{region "VFD"}
    //Status
    VTD_Control.Motor.Ready := (VTD_Control.Inputs.VFD_Status.%X0 OR VTD_Control.Inputs.VFD_Status.%X1) AND NOT VTD_Control.Motor.Error;
    VTD_Control.Motor.Error := VTD_Control.Inputs.VFD_Status.%X3 OR VTD_Control.Inputs.VFD_Status.%X7 OR NOT VTD_Control.Inputs.VFD_Status.%X13;
    VTD_Control.Motor.Enabled := VTD_Control.Inputs.VFD_Status.%X2;
    VTD_Control.Motor.Actual_Current := VTD_Control.Inputs.VFD_ActualCurrent;
    VTD_Control.Motor.Actual_Torque := SCALE_X(MIN := 0,
                                                VALUE := NORM_X(MIN := 0,
                                                                VALUE := VTD_Control.Inputs.VFD_ActualTorque,
                                                                MAX := 65536),
                                                MAX := 100);
    
    //Actual Speed
    IF MainSetpoint > 0 THEN
        VTD_Control.Motor.Speed_Actual := SCALE_X(MIN := 0,
                                                   VALUE := NORM_X(MIN := 0,
                                                                   VALUE := VTD_Control.Inputs.VFD_Speed_Actual,
                                                                   MAX := 16384),
                                                   MAX := 120);
        VTD_Control.Motor.Actual_Torque := SCALE_X(MIN := 0,
                                                    VALUE := NORM_X(MIN := 0,
                                                                    VALUE := VTD_Control.Inputs.VFD_ActualTorque * -1,
                                                                    MAX := 16384),
                                                    MAX := 100);
    ELSIF MainSetpoint < 0 THEN
        VTD_Control.Motor.Speed_Actual := SCALE_X(MIN := 0,
                                                   VALUE := NORM_X(MIN := 0,
                                                                   VALUE := VTD_Control.Inputs.VFD_Speed_Actual * -1,
                                                                   MAX := 16384),
                                                   MAX := 120);
        VTD_Control.Motor.Actual_Torque := SCALE_X(MIN := 0,
                                                    VALUE := NORM_X(MIN := 0,
                                                                    VALUE := VTD_Control.Inputs.VFD_ActualTorque * -1,
                                                                    MAX := 16384),
                                                    MAX := 100);
    ELSE
        VTD_Control.Motor.Speed_Actual := 0;
        VTD_Control.Motor.Actual_Torque := 0;
    END_IF;
    
    //SETPOINT
    IF VTD_Control.Motor_UP THEN
        MainSetpoint := SCALE_X(MIN := 0,
                                 VALUE := NORM_X(MIN := 0,
                                                 VALUE := VTD_Control.Motor_Speed,
                                                 MAX := 120),
                                 MAX := 1762);
    ELSIF VTD_Control.Motor_Down THEN
        MainSetpoint := (SCALE_X(MIN := 0,
                                  VALUE := NORM_X(MIN := 0,
                                                  VALUE := VTD_Control.Motor_Speed,
                                                  MAX := 120),
                                  MAX := 1762)) * -1;
    ELSE
        MainSetpoint := 0;
    END_IF;
    
    T_Setpoint_Delay(IN := MainSetpoint <> 0,
                          PT := T#0MS);
    
    IF T_Setpoint_Delay.Q THEN
        MainSetpoint1 := MainSetpoint;
    ELSE
        MainSetpoint1 := 0;
    END_IF;
    
    //Acceleration
    IF VTD_Control.Pallet_Loaded = 0 AND VTD_Control.Shuttle_Loaded = 0 THEN
        VTD_Control.Motor.Acc_Factor := SCALE_X(MIN := 0,
                                                 VALUE := NORM_X(MIN := 0,
                                                                 VALUE := 60.0,
                                                                 MAX := 100),
                                                 MAX := 16384);
    ELSIF Control.VTD_Order_Table[System_no].Pallet_Weight > 0 AND
        Control.VTD_Order_Table[System_no].Pallet_Weight <= "Settings_DB".VTD_Sys[System_no].Weight_Range_1 THEN
        VTD_Control.Motor.Acc_Factor := SCALE_X(MIN := 0,
                                                 VALUE := NORM_X(MIN := 0,
                                                                 VALUE := "Settings_DB".VTD_Sys[System_no].Acc_Range_1,
                                                                 MAX := 100),
                                                 MAX := 16384);
    ELSIF Control.VTD_Order_Table[System_no].Pallet_Weight > "Settings_DB".VTD_Sys[System_no].Weight_Range_1 AND
        Control_GVL.VTD_Order_Table[System_no].Pallet_Weight <= "Settings_DB".VTD_Sys[System_no].Weight_Range_2 THEN
        VTD_Control.Motor.Acc_Factor := SCALE_X(MIN := 0,
                                                 VALUE := NORM_X(MIN := 0,
                                                                 VALUE := "Settings_DB".VTD_Sys[System_no].Acc_Range_2,
                                                                 MAX := 100),
                                                 MAX := 16384);
    ELSIF Control.VTD_Order_Table[System_no].Pallet_Weight > "Settings_DB".VTD_Sys[System_no].Weight_Range_2 AND
        Control_GVL.VTD_Order_Table[System_no].Pallet_Weight <= "Settings_DB".VTD_Sys[System_no].Weight_Range_3 THEN
        VTD_Control.Motor.Acc_Factor := SCALE_X(MIN := 0,
                                                 VALUE := NORM_X(MIN := 0,
                                                                 VALUE := "Settings_DB".VTD_Sys[System_no].Acc_Range_3,
                                                                 MAX := 100),
                                                 MAX := 16384);
    ELSIF Control.VTD_Order_Table[System_no].Pallet_Weight > "Settings_DB".VTD_Sys[System_no].Weight_Range_3 OR
        Control_GVL.VTD_Order_Table[System_no].Pallet_Weight = 0 THEN
        VTD_Control.Motor.Acc_Factor := SCALE_X(MIN := 0,
                                                 VALUE := NORM_X(MIN := 0,
                                                                 VALUE := 100.0,
                                                                 MAX := 100),
                                                 MAX := 16384);
    ELSE
        VTD_Control.Motor.Acc_Factor := SCALE_X(MIN := 0,
                                                 VALUE := NORM_X(MIN := 0,
                                                                 VALUE := 100.0,
                                                                 MAX := 100),
                                                 MAX := 16384);
    END_IF;
    
    SinaSpeed(EnableAxis := VTD_Control.Motor_UP OR VTD_Control.Motor_Down,
              AckError := VTD_Control.Instruction.Reset OR "Reset_All" OR HMI_Reset,
              SpeedSp := MainSetpoint1,
              RefSpeed := 1762,
              HWIDSTW := VTD_Settings.G120_Hardware_ID,
              HWIDZSW := VTD_Settings.G120_Hardware_ID);
    
    //PARAMETERS
    //1082
    //2000
    //971
    //1820
{endregion}

HMI_Reset := (("Screen_DB_1".Reset_All[1] OR "VTD_HMI".Reset[1]) AND
("HMI_Box_Connected_1" = 11 AND "KEY REMOTE/LOCAL L1 - CH1(1)") OR
("HMI_Box_Connected_1" = 12 AND "KEY REMOTE/LOCAL L2 - CH1(1)") OR
("HMI_Box_Connected_1" = 13 AND "KEY REMOTE/LOCAL L3 - CH1(1)") OR
("HMI_Box_Connected_1" = 14 AND "KEY REMOTE/LOCAL L4 - CH1(1)") OR
("HMI_Box_Connected_1" = 15 AND "KEY REMOTE/LOCAL L5 - CH1(1)") OR
("HMI_Box_Connected_1" = 16 AND "KEY REMOTE/LOCAL L6 - CH1(1)") OR
("HMI_Box_Connected_1" = 21 AND "KEY REMOTE/LOCAL L1 - CH1(2)") OR
("HMI_Box_Connected_1" = 22 AND "KEY REMOTE/LOCAL L2 - CH1(2)") OR
("HMI_Box_Connected_1" = 23 AND "KEY REMOTE/LOCAL L3 - CH1(2)") OR
("HMI_Box_Connected_1" = 24 AND "KEY REMOTE/LOCAL L4 - CH1(2)") OR
("HMI_Box_Connected_1" = 25 AND "KEY REMOTE/LOCAL L5 - CH1(2)") OR
("HMI_Box_Connected_1" = 26 AND "KEY REMOTE/LOCAL L6 - CH1(2)"))
OR
(("Screen_DB_1".Reset_All[2] OR "VTD_HMI".Reset[2]) AND
("HMI_Box_Connected_2" = 11 AND "KEY REMOTE/LOCAL L1 - CH1(1)") OR
("HMI_Box_Connected_2" = 12 AND "KEY REMOTE/LOCAL L2 - CH1(1)") OR
("HMI_Box_Connected_2" = 13 AND "KEY REMOTE/LOCAL L3 - CH1(1)") OR
("HMI_Box_Connected_2" = 14 AND "KEY REMOTE/LOCAL L4 - CH1(1)") OR
("HMI_Box_Connected_2" = 15 AND "KEY REMOTE/LOCAL L5 - CH1(1)") OR
("HMI_Box_Connected_2" = 16 AND "KEY REMOTE/LOCAL L6 - CH1(1)") OR
("HMI_Box_Connected_2" = 21 AND "KEY REMOTE/LOCAL L1 - CH1(2)") OR
("HMI_Box_Connected_2" = 22 AND "KEY REMOTE/LOCAL L2 - CH1(2)") OR
("HMI_Box_Connected_2" = 23 AND "KEY REMOTE/LOCAL L3 - CH1(2)") OR
("HMI_Box_Connected_2" = 24 AND "KEY REMOTE/LOCAL L4 - CH1(2)") OR
("HMI_Box_Connected_2" = 25 AND "KEY REMOTE/LOCAL L5 - CH1(2)") OR
("HMI_Box_Connected_2" = 26 AND "KEY REMOTE/LOCAL L6 - CH1(2)"));

//Assign local vars to outputs
VTD_Control.Outputs.LP1_Retract := DP1_Retract;
VTD_Control.Outputs.LP1_Extend := DP1_Extend;
VTD_Control.Outputs.LP2_Retract := DP2_Retract;
VTD_Control.Outputs.LP2_Extend := DP2_Extend;

END_FUNCTION_BLOCK
